// TIA Portal project "HeatCt1_4S" (V13)

(* hardware
DEVICE "S7300/ET200M-Station_1"  S7-300 station
   slot 0: "Profilschiene_0"  Rail  6ES7 390-1***0-0AA0
   slot 1: "PS 307 5A_1"  PS 307 5A  6ES7 307-1EA00-0AA0
   slot 2: "SIMATIC S7-300"  CPU 314C-2 PN/DP  6ES7 314-6EH04-0AB0  V3.3
      slot 2: "PROFINET-Schnittstelle_1"  PN-IO
         slot 1: "Port_1"  Port
         slot 2: "Port_2"  Port
      slot 5: "DI 24/DO 16_1"  DI24/DO16
      slot 6: "AI 5/AO 2_1"  AI5/AO2
      slot 7: "Zählen_1"  Counter
      slot 8: "Positionieren_1"  Positioning
   slot 4: "CP 343-2_1"  CP 343-2  6GK7 343-2AH01-0XA0  V3.1
*)

// ===== PLC "SIMATIC S7-300"  CPU 314C-2 PN/DP =====

VAR_GLOBAL   // PLC tag table "Standard-Variablentabelle"
   "Mx_Clock10Hz" AT %M100.0 : Bool;   // CPU clock memory-flag 0: f = 10 Hz / T = 0,1 s
   "Mx_Clock5Hz" AT %M100.1 : Bool;   // CPU clock memory-flag 1: f = 5 Hz / T = 0,2 s
   "Mx_Clock2,5Hz" AT %M100.2 : Bool;   // CPU clock memory-flag 2: f = 2,5 Hz / T = 0,4 s
   "Mx_Clock2Hz" AT %M100.3 : Bool;   // CPU clock memory-flag 3: f = 2 Hz / T = 0,5 s
   "Mx_Clock1,25Hz" AT %M100.4 : Bool;   // CPU clock memory-flag 4: f = 1,25 Hz / T = 0,8 s
   "Mx_Clock1Hz" AT %M100.5 : Bool;   // CPU clock memory-flag 5: f = 1 Hz / T = 1 s
   "Mx_Clock0,625Hz" AT %M100.6 : Bool;   // CPU clock memory-flag 6: f = 0,625 Hz / T = 1,6 s
   "Mx_Clock0,5Hz" AT %M100.7 : Bool;   // CPU clock memory-flag 7: f = 0,5 Hz / T = 2 s
   "C1_RadiatorCounter" AT %C1 : Counter;   // Counter to count the number of radiators
   "Ix_S0_SystemOFF" AT %I124.0 : Bool;   // Heating system off (NC)
   "Ix_S1_SystemON" AT %I124.1 : Bool;   // Heating system on (stand-by mode)
   "Ix_S2_RadiatorsON" AT %I124.2 : Bool;   // Switch on any of the radiators
   "Ix_S3_RadiatorsOFF" AT %I124.3 : Bool;   // Switch off any of the radiators (NC)
   "Mx_Step1" AT %M1.0 : Bool;   // Grafcet, step-flag 1
   "Mx_Step2" AT %M1.1 : Bool;   // Grafcet, step-flag 2
   "Mx_PEdgeFlag_Step1" AT %M1.2 : Bool;   // Positive edge flag is activated when step 1 is activated
   "Mx_StartingFlag" AT %M2.0 : Bool;   // Starting flag to activate the sequence (step 1)
   "Mx_LockCounter" AT %M10.0 : Bool;   // The counter must be locked as soon as all 4 radiators are active
   "Mx_PEdgeFlag_S2" AT %M10.1 : Bool;   // Positive edge flag is activated on pressing S2
   "Mx_PEdgeFlag_S3" AT %M10.2 : Bool;   // Positive edge flag is activated on pressing S3
   "Mb_FlagByte1" AT %MB1 : Byte;   // Flag byte 1
   "Md_AnalogOut" AT %MD18 : Real;   // Result of the scaling
   "Md_AnalogOutRound1" AT %MD26 : DInt;   // Scaled analog value rounded to an integer (32-Bit)
   "Mw_CountValueWORD" AT %MW12 : Word;   // Count value in the format WORD
   "Mw_ReturnValue" AT %MW22 : Word;   // Returns the value to 0 if the scaling works correctly
   "Mw_AnalogOutRound2" AT %MW30 : Int;   // Scaled analog value rounded to an integer (16-Bit)
   "Iw_S4_RadiatorsONOFF" AT %IW752 : Int;   // Switch on/off any of the radiators (analog)
   "Qx_P40_Radiator4Active_ASi" AT %Q87.4 : Bool;   // Storage area: Radiator 4 is active (slave address 22)
   "Qx_P30_Radiator3Active_ASi" AT %Q87.5 : Bool;   // Storage area: Radiator 3 is active (slave address 22)
   "Qx_P20_Radiator2Active_ASi" AT %Q87.6 : Bool;   // Storage area: Radiator 2 is active (slave address 22)
   "Qx_P10_Radiator1Active_ASi" AT %Q87.7 : Bool;   // Storage area: Radiator 1 is active (slave address 22)
   "Qx_Q1_FeedRadiator1" AT %Q124.0 : Bool;   // Positioning valve Q1, feed radiator 1
   "Qx_Q2_FeedRadiator2" AT %Q124.1 : Bool;   // Positioning valve Q2, feed radiator 2
   "Qx_Q3_FeedRadiator3" AT %Q124.2 : Bool;   // Positioning valve Q3, feed radiator 3
   "Qx_Q4_FeedRadiator4" AT %Q124.3 : Bool;   // Positioning valve Q4, feed radiator 4
   "Qx_P1_SystemON" AT %Q125.0 : Bool;   // Heating system in stand-by mode
   "Qx_P10_Radiator1Active" AT %Q125.4 : Bool;   // Radiator 1 is active
   "Qx_P20_Radiator2Active" AT %Q125.5 : Bool;   // Radiator 2 is active
   "Qx_P30_Radiator3Active" AT %Q125.6 : Bool;   // Radiator 3 is active
   "Qx_P40_Radiator4Active" AT %Q125.7 : Bool;   // Radiator 4 is active
   "Qb_Radiators" AT %QB124 : Byte;   // Outputbyte, the radiators are connected to
END_VAR

ORGANIZATION_BLOCK "Main"   // OB1, FBD
TITLE = "Main Program Sweep (Cycle)"
{ S7_Optimized_Access := 'FALSE' }
VERSION : 0.1
BEGIN
END_ORGANIZATION_BLOCK

ORGANIZATION_BLOCK "COMPLETE RESTART"   // OB100, FBD
TITLE = "Complete Restart"
{ S7_Optimized_Access := 'FALSE' }
VERSION : 0.1
BEGIN

REGION Network 1: Reset flag byte 1 (step-flags)
   // With the instruction "MOVE", all bits of memory flag byte number 1 will be overwritten with the value 0. Thus it is guaranteed that all steps are deactivated when the status of the PLC changes from RUN to STOP and back to RUN. Otherwise the plant will go back to the previous status without activating any pushbuttons.
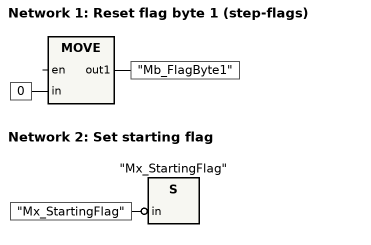
   "Mb_FlagByte1" := 0;
END_REGION

REGION Network 2: Set starting flag
   IF NOT "Mx_StartingFlag" THEN "Mx_StartingFlag" := TRUE; END_IF;
END_REGION
END_ORGANIZATION_BLOCK